PROGRAM Q1_MOTOR
VAR
	ClearFault: FB_ClearFault;
	SetEnableState: FB_SetEnableState;
	SetHomingParameter: FB_SetHomingParameter;
	FindHome: FB_FindHome;
	SetMotorParameter: FB_SetMotorParameter;
	SetPositionProfile: FB_SetPositionProfile;
	SetOperationMode: FB_SetOperationMode;
	MoveToPosition: FB_MoveToPosition;
	GetMovementState: FB_GetMovementState;
	SetDisableState: FB_SetDisableState;
	SetPositionMust: FB_SetPositionMust;
	POSITION: DINT;
END_VAR

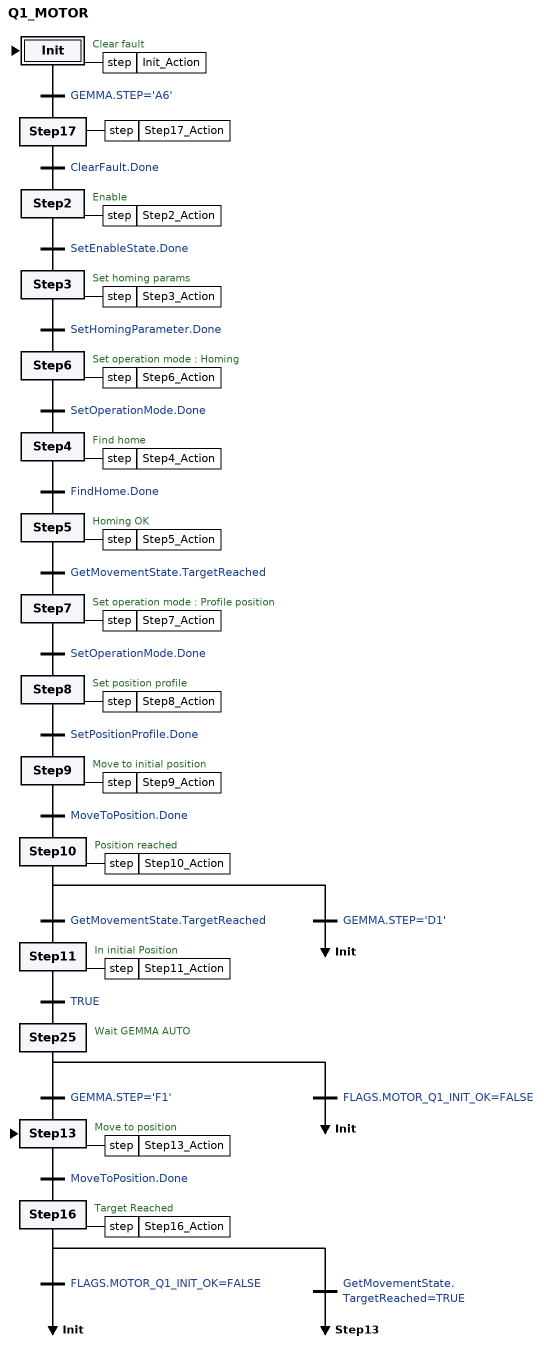
// Clear fault
INITIAL_STEP Init:
    Init_Action(N);  // step action
END_STEP
TRANSITION FROM Init TO Step17
    := GEMMA.STEP='A6';
END_TRANSITION
STEP Step17:
    Step17_Action(N);  // step action
END_STEP
TRANSITION FROM Step17 TO Step2
    := ClearFault.Done;
END_TRANSITION
// Enable
STEP Step2:
    Step2_Action(N);  // step action
END_STEP
TRANSITION FROM Step2 TO Step3
    := SetEnableState.Done;
END_TRANSITION
// Set homing params
STEP Step3:
    Step3_Action(N);  // step action
END_STEP
TRANSITION FROM Step3 TO Step6
    := SetHomingParameter.Done;
END_TRANSITION
// Set operation mode : Homing
STEP Step6:
    Step6_Action(N);  // step action
END_STEP
TRANSITION FROM Step6 TO Step4
    := SetOperationMode.Done;
END_TRANSITION
// Find home
STEP Step4:
    Step4_Action(N);  // step action
END_STEP
TRANSITION FROM Step4 TO Step5
    := FindHome.Done;
END_TRANSITION
// Homing OK
STEP Step5:
    Step5_Action(N);  // step action
END_STEP
TRANSITION FROM Step5 TO Step7
    := GetMovementState.TargetReached;
END_TRANSITION
// Set operation mode : Profile position
STEP Step7:
    Step7_Action(N);  // step action
END_STEP
TRANSITION FROM Step7 TO Step8
    := SetOperationMode.Done;
END_TRANSITION
// Set position profile
STEP Step8:
    Step8_Action(N);  // step action
END_STEP
TRANSITION FROM Step8 TO Step9
    := SetPositionProfile.Done;
END_TRANSITION
// Move to initial position
STEP Step9:
    Step9_Action(N);  // step action
END_STEP
TRANSITION FROM Step9 TO Step10
    := MoveToPosition.Done;
END_TRANSITION
// Position reached
STEP Step10:
    Step10_Action(N);  // step action
END_STEP
TRANSITION FROM Step10 TO Step11
    := GetMovementState.TargetReached;
END_TRANSITION
TRANSITION FROM Step10 TO Init
    := GEMMA.STEP='D1';
END_TRANSITION
// In initial Position
STEP Step11:
    Step11_Action(N);  // step action
END_STEP
TRANSITION FROM Step11 TO Step25
    := TRUE;
END_TRANSITION
// Wait GEMMA AUTO
STEP Step25:
END_STEP
TRANSITION FROM Step25 TO Step13
    := GEMMA.STEP='F1';
END_TRANSITION
TRANSITION FROM Step25 TO Init
    := FLAGS.MOTOR_Q1_INIT_OK=FALSE;
END_TRANSITION
// Move to position
STEP Step13:
    Step13_Action(N);  // step action
END_STEP
TRANSITION FROM Step13 TO Step16
    := MoveToPosition.Done;
END_TRANSITION
// Target Reached
STEP Step16:
    Step16_Action(N);  // step action
END_STEP
TRANSITION FROM Step16 TO Init
    := FLAGS.MOTOR_Q1_INIT_OK=FALSE;
END_TRANSITION
TRANSITION FROM Step16 TO Step13
    := GetMovementState.TargetReached=TRUE;
END_TRANSITION

ACTION Step5_Action:
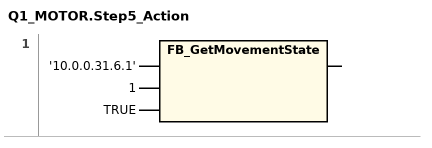
// NETWORK 1
FB_GetMovementState('10.0.0.31.6.1', 1, TRUE);
END_ACTION

ACTION Step16_Action:
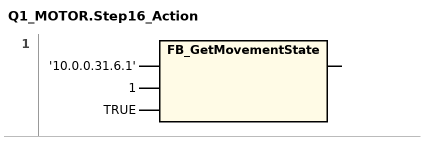
// NETWORK 1
FB_GetMovementState('10.0.0.31.6.1', 1, TRUE);
END_ACTION

ACTION Step7_Action:
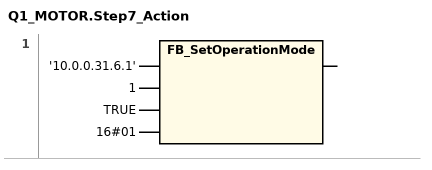
// NETWORK 1
FB_SetOperationMode('10.0.0.31.6.1', 1, TRUE, 16#01);
END_ACTION

ACTION Step2_Action:
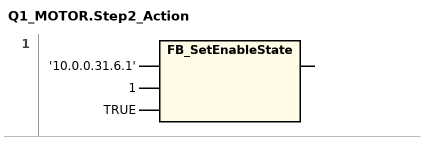
// NETWORK 1
FB_SetEnableState('10.0.0.31.6.1', 1, TRUE);
END_ACTION

ACTION Step17_Action:
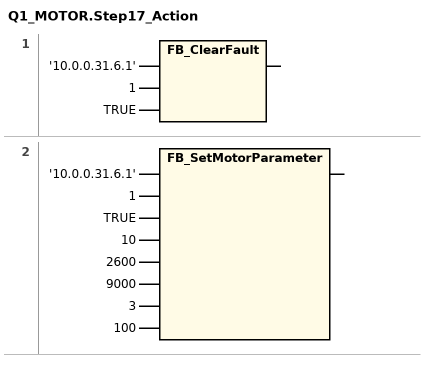
// NETWORK 1
FB_ClearFault('10.0.0.31.6.1', 1, TRUE);

// NETWORK 2
FB_SetMotorParameter('10.0.0.31.6.1', 1, TRUE, 10, 2600, 9000, 3, 100);
END_ACTION

ACTION Step6_Action:
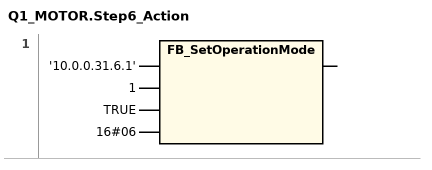
// NETWORK 1
FB_SetOperationMode('10.0.0.31.6.1', 1, TRUE, 16#06);
END_ACTION

ACTION Step13_Action:
(*Limitation deplacement Moteur*)
IF FLAGS.MOTOR_Q1_POSITION>MOTOR_Q1_POSITION_MAX THEN
	POSITION:=MOTOR_Q1_POSITION_MAX;
ELSIF FLAGS.MOTOR_Q1_POSITION<0 THEN
	POSITION:=0;
ELSE
	POSITION:=FLAGS.MOTOR_Q1_POSITION;
END_IF


MoveToPosition(
	ADSNetId:= '10.0.0.31.6.1',
	NodeId:= 1,
	Write:= TRUE,
	TargetPosition:= POSITION,
	Absolut:= TRUE);
END_ACTION

ACTION Step10_Action:
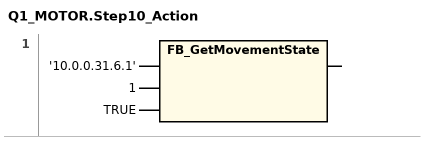
// NETWORK 1
FB_GetMovementState('10.0.0.31.6.1', 1, TRUE);
END_ACTION

ACTION Step3_Action:
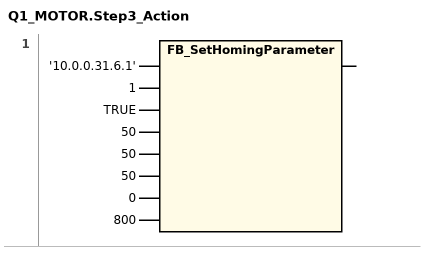
// NETWORK 1
FB_SetHomingParameter('10.0.0.31.6.1', 1, TRUE, 50, 50, 50, 0, 800);
END_ACTION

ACTION Step9_Action:
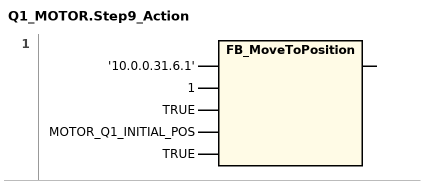
// NETWORK 1
FB_MoveToPosition('10.0.0.31.6.1', 1, TRUE, MOTOR_Q1_INITIAL_POS, TRUE);
END_ACTION

ACTION Step8_Action:
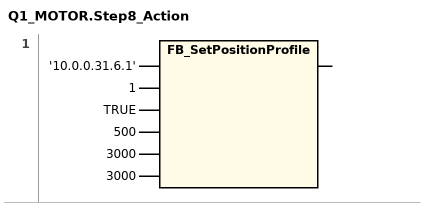
// NETWORK 1
FB_SetPositionProfile('10.0.0.31.6.1', 1, TRUE, 500, 3000, 3000);
END_ACTION

ACTION Step11_Action:

(*SetDisableState(
	ADSNetId:= '10.0.0.31.6.1',
	NodeId:= 1,
	Write:= TRUE);*)

FLAGS.MOTOR_Q1_INIT_OK:=TRUE;
END_ACTION

ACTION Init_Action:

END_ACTION

ACTION Step4_Action:
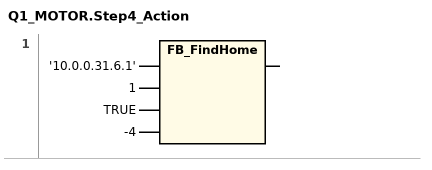
// NETWORK 1
FB_FindHome('10.0.0.31.6.1', 1, TRUE, -4);
END_ACTION

END_PROGRAM

(* stored: Version 1.1.0.1, ProductVersion 3.1.0.26
   POU Q1_MOTOR: Id {f755a67c-d6ae-47de-85f7-bd33b247bdee}
   Action Step5_Action: Id {107c0bbb-6a26-454a-b059-6dfd13c1a286}
   Action Step16_Action: Id {1b26b01d-ba6f-4a3f-94f2-c29ee05dcabd}
   Action Step7_Action: Id {2f082169-a36b-4af5-97f0-1e632a444508}
   Action Step2_Action: Id {60f21950-58e5-4e1f-9be2-173d18be152b}
   Action Step17_Action: Id {61f07674-dc03-493d-9287-5d3d53586e2e}
   Action Step6_Action: Id {70ab760f-b945-4cef-86b2-b6da8261c89b}
   Action Step13_Action: Id {86cf10b8-7a87-4ef2-b969-08524a2ff05f}
   Action Step10_Action: Id {9df29495-2113-4b27-a29d-2b56796038a0}
   Action Step3_Action: Id {b0343ce0-4ec2-44c1-b097-8f082237a3e5}
   Action Step9_Action: Id {c296f40d-1d46-4684-88c9-373a6a7bade1}
   Action Step8_Action: Id {c9f12793-d210-4c52-b204-61cc728fd1f2}
   Action Step11_Action: Id {dd99d647-7a7b-4f34-96ce-dae9b7a99168}
   Action Init_Action: Id {e08471ac-ff90-4160-8086-597a2d33ce5b}
   Action Step4_Action: Id {f52bcb0c-2b6b-46b8-aebe-076d130abcb9} *)
